{attribute addProperty BoxType "KL3162"}
{attribute addProperty Id "Channel_1Channel_585D17BE00Channel_2Channel_585D17BE00"}
{attribute addProperty CRC "3457887495"}
{attribute addProperty SizeInBites "0"}
{attribute addProperty SizeInBytes "0"}
TYPE KL3162_CE1B2D07 :
STRUCT
	{attribute addProperty Name "Channel_1"}
	Channel_1 : Channel_585D17BE;
	{attribute addProperty Name "Channel_2"}
	Channel_2 : Channel_585D17BE;
END_STRUCT
END_TYPE

(* stored: Version 1.2.0.0, ProductVersion 3.1.4024.9
   DUT KL3162_CE1B2D07: Id {ce7e6645-c581-41c6-9c90-917ff8124946} *)
